Staubli VAL3: checkTaskStates.pgx

program checkTaskStates(num& nTaskState_[])
  local num idx
  local string sText
  local num count
  local string callStack[20]
  local num line
  local string library
  local string program
  local string code
begin
    //\brief
  //
  //\change
  //07.06.06, vdg: log status of user tasks
  // go through list of tasks
  //\var idx
  //\var sText
  //\var count
  //\var callStack
  //\var line
  //\var library
  //\var program
  //\var code
  //\param nTaskState_
  //
//!change 07.06.06, vdg: log status of user tasks
  // go through list of tasks
  for idx=0 to size(sTaskName)-1
    // check if task state has changed
    if taskStatus(sTaskName[idx])!=nTaskState_[idx]
      // store new task state
      nTaskState_[idx]=taskStatus(sTaskName[idx])
      // get message string
      call ui:getTaskErrorMsg(nTaskState_[idx],sText)
      // log the message
      logMsg(sTaskName[idx]+": "+sText)
    endIf
    // get call stack of task
    count=$taskCallStack(sTaskName[idx],callStack)
    if idx==1
      call parseStackInfo(callStack,library,program,line,code)
      if program=="SP_Traj"
        call list:resizeString(programList,max(size(programList),line))
        programList[line]=code
      endIf
    endIf
    if count>0
      stat:sTaskStack[idx]=callStack[count-1]
    else
      stat:sTaskStack[idx]=""
    endIf
  endFor
  // check if home return is active
  //!change vdg, 11.03.08 : set SYS:bHomeRetActive when home return task exists, not only when it is executing
  SYS:bHomeRetActive=taskStatus(sTaskName[2])!=-1
  //
  //!issue 22
  // poll state of user PLC
  call prg:statusPLC(stat:PLCStatus,stat:PLCStatusText)
end
